(*
Returns the index of the task that calls this function.

..note:: Falls back to task index 1 if  called outside the real-time context.
*)
FUNCTION F_GetCurrentTaskIndex : DINT
VAR
	fbGetCurrentTaskIndex : Tc2_System.GETCURTASKINDEX;
END_VAR

fbGetCurrentTaskIndex();
F_GetCurrentTaskIndex := fbGetCurrentTaskIndex.Index;

END_FUNCTION

(* stored: Version 1.1.0.1
   POU F_GetCurrentTaskIndex: Id {9290cc24-abd2-03dc-065e-9ac4c762564f}, SpecialFunc None *)
